{attribute addProperty BoxType "EL3681-0000-0021"}
{attribute addProperty Id "SAI_InputsAT %I*SAI_Inputs_166EE3574860SAI_FeedbackAT %I*SAI_Feedback_DF9848341620SAI_RangeAT %Q*SAI_Range_80D0ED7D1620WcStateAT %I*WcState_F855686C1620InfoDataAT %I*InfoData_BC63D37F80100"}
{attribute addProperty CRC "757688760"}
{attribute addProperty SizeInBites "176"}
{attribute addProperty SizeInBytes "22"}
TYPE EL3681_01269A60 :
STRUCT
	{attribute addProperty Name "SAI_Inputs"}
	SAI_Inputs : SAI_Inputs_166EE357;
	{attribute addProperty Name "SAI_Feedback"}
	SAI_Feedback : SAI_Feedback_DF984834;
	{attribute addProperty Name "SAI_Range"}
	SAI_Range : SAI_Range_80D0ED7D;
	{attribute addProperty Name "WcState"}
	WcState : WcState_F855686C;
	{attribute addProperty Name "InfoData"}
	InfoData : InfoData_BC63D37F;
END_STRUCT
END_TYPE

(* stored: Version 1.2.0.0, ProductVersion 3.1.4024.9
   DUT EL3681_01269A60: Id {6185ae4e-2166-4f19-9c05-6a620d30d51f} *)
